TYPE ST_P2AxisName :   //2#部分轴
STRUCT
P2M1_AnCarryingLine	:INT:=1;	//1号叠台	正极送片搬运平移 
P2M1_AnCarryingUpDown	:INT:=2;	//1号叠台	正极送片搬运升降
P2M1_AnCarryingWhirling	:INT:=3;	//1号叠台	正极送片搬运旋转
P2M1_AnDTCarryingLine	:INT:=4;	//1号叠台	正极叠台搬运平移1
P2M1_AnDTCarryingUpDown	:INT:=5;	//1号叠台	正极叠台搬运升降
P2M1_AndeviationX1	:INT:=6;	//1号叠台	正极纠偏平台X1
P2M1_AndeviationX2	:INT:=7;	//1号叠台	正极纠偏平台X2
P2M1_AndeviationY	:INT:=8;	//1号叠台	正极纠偏平台Y
P2M1_CaCarryingLine1	:INT:=9;	//1号叠台	负极送片搬运1平移
P2M1_CaCarryingUpDown1	:INT:=10;	//1号叠台	负极送片搬运1升降
P2M1_CaCarryingWhirling1	:INT:=11;	//1号叠台	负极送片搬运1旋转
P2M1_CaCarryingLine2	:INT:=12;	//1号叠台	负极送片搬运2平移
P2M1_CaCarryingUpDown2	:INT:=13;	//1号叠台	负极送片搬运2升降
P2M1_CaBelt	:INT:=14;	//1号叠台	负极送片皮带
P2M1_CaDTCarryingLine	:INT:=15;	//1号叠台	负极叠台搬运平移
P2M1_CaDTCarryingUpDown	:INT:=16;	//1号叠台	负极叠台搬运升降
P2M1_CadeviationX1	:INT:=17;	//1号叠台	负极纠偏平台X1
P2M1_CadeviationX2	:INT:=18;	//1号叠台	负极纠偏平台X2
P2M1_CadeviationY	:INT:=19;	//1号叠台	负极纠偏平台Y
P2M1_SEPTAunwinding	:INT:=20;	//1号叠台	隔膜放卷
P2M1_SEPTAdeviation1	:INT:=21;	//1号叠台	隔膜放卷纠偏
P2M1_SEPTAdeviation2	:INT:=22;	//1号叠台	隔膜尾部纠偏
P2M1_SEPTATension	:INT:=23;	//1号叠台	隔膜摆杆张力
P2M1_SEPTATCache	:INT:=24;	//1号叠台	隔膜缓存
P2M1_SEPTATLine	:INT:=25;	//1号叠台	隔膜平移
P2M1_DTUpDown	:INT:=26;	//1号叠台	叠台升降
P2M1_LeftYDLine	:INT:=27;	//1号叠台	左压刀开合
P2M1_LeftYDUpDown	:INT:=28;	//1号叠台	左压刀升降
P2M1_RightYDLine	:INT:=29;	//1号叠台	右压刀开合
P2M1_RightYDUpDown	:INT:=30;	//1号叠台	右压刀升降
P2M1_TailCurlLine	:INT:=31;	//1号叠台	尾卷夹电芯平移
P2M1_TailCurlUpDown	:INT:=32;	//1号叠台	尾卷夹电芯升降
P2M1_TailCurlRetracting	:INT:=33;	//1号叠台	尾卷夹电芯伸缩
P2M1_TailCurlWhirling	:INT:=34;	//1号叠台	尾卷夹电芯旋转
P2M1_TailCurlSEPTALine	:INT:=35;	//1号叠台	夹膜平移
P2M1_TailCurlSEPTAUpDown	:INT:=36;	//1号叠台	夹膜升降
P2M1_LCurlingneedleLine	:INT:=37;	//1号叠台	长卷针平移
P2M1_SCurlingneedleLine	:INT:=38;	//1号叠台	短卷针平移
P2M1_LCurlingneedleWhirling	:INT:=39;	//1号叠台	长卷针旋转
P2M1_SCurlingneedleWhirling	:INT:=40;	//1号叠台	短卷针旋转
P2M1_GluingLine	:INT:=41;	//1号叠台	侧贴夹平移
P2M1_GluingWhirling	:INT:=42;	//1号叠台	侧贴夹旋转
P2M1_GluingRetracting	:INT:=43;	//1号叠台	贴胶头进退
P2M1_GluingUpDown	:INT:=44;	//1号叠台	拉胶升降
P2M1_Standby1	:INT:=45;	//1号叠台	备用
P2M1_Standby2	:INT:=46;	//1号叠台	备用

P2M2_AnCarryingLine	:INT:=47;	//2号叠台	正极送片搬运平移
P2M2_AnCarryingUpDown	:INT:=48;	//2号叠台	正极送片搬运升降
P2M2_AnCarryingWhirling	:INT:=49;	//2号叠台	正极送片搬运旋转
P2M2_AnDTCarryingLine	:INT:=50;	//2号叠台	正极叠台搬运平移
P2M2_AnDTCarryingUpDown	:INT:=51;	//2号叠台	正极叠台搬运升降
P2M2_AndeviationX1	:INT:=52;	//2号叠台	正极纠偏平台X1
P2M2_AndeviationX2	:INT:=53;	//2号叠台	正极纠偏平台X2
P2M2_AndeviationY	:INT:=54;	//2号叠台	正极纠偏平台Y
P2M2_CaCarryingLine1	:INT:=55;	//2号叠台	负极送片搬运1平移
P2M2_CaCarryingUpDown1	:INT:=56;	//2号叠台	负极送片搬运1升降
P2M2_CaCarryingWhirling1	:INT:=57;	//2号叠台	负极送片搬运1旋转
P2M2_CaCarryingLine2	:INT:=58;	//2号叠台	负极送片搬运2平移
P2M2_CaCarryingUpDown2	:INT:=59;	//2号叠台	负极送片搬运2升降
P2M2_CaBelt	:INT:=60;	//2号叠台	负极送片皮带
P2M2_CaDTCarryingLine	:INT:=61;	//2号叠台	负极叠台搬运平移
P2M2_CaDTCarryingUpDown	:INT:=62;	//2号叠台	负极叠台搬运升降
P2M2_CadeviationX1	:INT:=63;	//2号叠台	负极纠偏平台X1
P2M2_CadeviationX2	:INT:=64;	//2号叠台	负极纠偏平台X2
P2M2_CadeviationY	:INT:=65;	//2号叠台	负极纠偏平台Y
P2M2_SEPTAunwinding	:INT:=66;	//2号叠台	隔膜放卷
P2M2_SEPTAdeviation1	:INT:=67;	//2号叠台	隔膜放卷纠偏
P2M2_SEPTAdeviation2	:INT:=68;	//2号叠台	隔膜尾部纠偏
P2M2_SEPTATension	:INT:=69;	//2号叠台	隔膜摆杆张力
P2M2_SEPTATCache	:INT:=70;	//2号叠台	隔膜缓存
P2M2_SEPTATLine	:INT:=71;	//2号叠台	隔膜平移
P2M2_DTUpDown	:INT:=72;	//2号叠台	叠台升降
P2M2_LeftYDLine	:INT:=73;	//2号叠台	左压刀开合
P2M2_LeftYDUpDown	:INT:=74;	//2号叠台	左压刀升降
P2M2_RightYDLine	:INT:=75;	//2号叠台	右压刀开合
P2M2_RightYDUpDown	:INT:=76;	//2号叠台	右压刀升降
P2M2_TailCurlLine	:INT:=77;	//2号叠台	尾卷夹电芯平移
P2M2_TailCurlUpDown	:INT:=78;	//2号叠台	尾卷夹电芯升降
P2M2_TailCurlRetracting	:INT:=79;	//2号叠台	尾卷夹电芯伸缩
P2M2_TailCurlWhirling	:INT:=80;	//2号叠台	尾卷夹电芯旋转
P2M2_TailCurlSEPTALine	:INT:=81;	//2号叠台	夹膜平移
P2M2_TailCurlSEPTAUpDown	:INT:=82;	//2号叠台	夹膜升降
P2M2_LCurlingneedleLine	:INT:=83;	//2号叠台	长卷针平移
P2M2_SCurlingneedleLine	:INT:=84;	//2号叠台	短卷针平移
P2M2_LCurlingneedleWhirling	:INT:=85;	//2号叠台	长卷针旋转
P2M2_SCurlingneedleWhirling	:INT:=86;	//2号叠台	短卷针旋转
P2M2_GluingLine	:INT:=87;	//2号叠台	侧贴夹平移
P2M2_GluingWhirling	:INT:=88;	//2号叠台	侧贴夹旋转
P2M2_GluingRetracting	:INT:=89;	//2号叠台	贴胶头进退
P2M2_GluingUpDown	:INT:=90;	//2号叠台	拉胶升降
P2M2_Standby1	:INT:=91;	//2号叠台	备用
P2M2_Standby2	:INT:=92;	//2号叠台	备用

P2M3_AnCarryingLine	:INT:=93;	//3号叠台	正极送片搬运平移
P2M3_AnCarryingUpDown	:INT:=94;	//3号叠台	正极送片搬运升降
P2M3_AnCarryingWhirling	:INT:=95;	//3号叠台	正极送片搬运旋转
P2M3_AnDTCarryingLine	:INT:=96;	//3号叠台	正极叠台搬运平移
P2M3_AnDTCarryingUpDown	:INT:=97;	//3号叠台	正极叠台搬运升降
P2M3_AndeviationX1	:INT:=98;	//3号叠台	正极纠偏平台X1
P2M3_AndeviationX2	:INT:=99;	//3号叠台	正极纠偏平台X2
P2M3_AndeviationY	:INT:=100;	//3号叠台	正极纠偏平台Y
P2M3_CaCarryingLine1	:INT:=101;	//3号叠台	负极送片搬运1平移
P2M3_CaCarryingUpDown1	:INT:=102;	//3号叠台	负极送片搬运1升降
P2M3_CaCarryingWhirling1	:INT:=103;	//3号叠台	负极送片搬运1旋转
P2M3_CaCarryingLine2	:INT:=104;	//3号叠台	负极送片搬运2平移
P2M3_CaCarryingUpDown2	:INT:=105;	//3号叠台	负极送片搬运2升降
P2M3_CaBelt	:INT:=106;	//3号叠台	负极送片皮带
P2M3_CaDTCarryingLine	:INT:=107;	//3号叠台	负极叠台搬运平移
P2M3_CaDTCarryingUpDown	:INT:=108;	//3号叠台	负极叠台搬运升降
P2M3_CadeviationX1	:INT:=109;	//3号叠台	负极纠偏平台X1
P2M3_CadeviationX2	:INT:=110;	//3号叠台	负极纠偏平台X2
P2M3_CadeviationY	:INT:=111;	//3号叠台	负极纠偏平台Y
P2M3_SEPTAunwinding	:INT:=112;	//3号叠台	隔膜放卷
P2M3_SEPTAdeviation1	:INT:=113;	//3号叠台	隔膜放卷纠偏
P2M3_SEPTAdeviation2	:INT:=114;	//3号叠台	隔膜尾部纠偏
P2M3_SEPTATension	:INT:=115;	//3号叠台	隔膜摆杆张力
P2M3_SEPTATCache	:INT:=116;	//3号叠台	隔膜缓存
P2M3_SEPTATLine	:INT:=117;	//3号叠台	隔膜平移
P2M3_DTUpDown	:INT:=118;	//3号叠台	叠台升降
P2M3_LeftYDLine	:INT:=119;	//3号叠台	左压刀开合
P2M3_LeftYDUpDown	:INT:=120;	//3号叠台	左压刀升降
P2M3_RightYDLine	:INT:=121;	//3号叠台	右压刀开合
P2M3_RightYDUpDown	:INT:=122;	//3号叠台	右压刀升降
P2M3_TailCurlLine	:INT:=123;	//3号叠台	尾卷夹电芯平移
P2M3_TailCurlUpDown	:INT:=124;	//3号叠台	尾卷夹电芯升降
P2M3_TailCurlRetracting	:INT:=125;	//3号叠台	尾卷夹电芯伸缩
P2M3_TailCurlWhirling	:INT:=126;	//3号叠台	尾卷夹电芯旋转
P2M3_TailCurlSEPTALine	:INT:=127;	//3号叠台	夹膜平移
P2M3_TailCurlSEPTAUpDown	:INT:=128;	//3号叠台	夹膜升降
P2M3_LCurlingneedleLine	:INT:=129;	//3号叠台	长卷针平移
P2M3_SCurlingneedleLine	:INT:=130;	//3号叠台	短卷针平移
P2M3_LCurlingneedleWhirling	:INT:=131;	//3号叠台	长卷针旋转
P2M3_SCurlingneedleWhirling	:INT:=132;	//3号叠台	短卷针旋转
P2M3_GluingLine	:INT:=133;	//3号叠台	侧贴夹平移
P2M3_GluingWhirling	:INT:=134;	//3号叠台	侧贴夹旋转
P2M3_GluingRetracting	:INT:=135;	//3号叠台	贴胶头进退
P2M3_GluingUpDown	:INT:=136;	//3号叠台	拉胶升降
P2M3_Standby1	:INT:=137;	//3号叠台	备用
P2M3_Standby2	:INT:=138;	//3号叠台	备用


END_STRUCT
END_TYPE

(* stored: Version 1.1.0.1, ProductVersion 3.1.4024.9
   DUT ST_P2AxisName: Id {b7d17884-a1af-476a-b448-6ef5a02acace} *)
